//{attribute 'qualified_only'}
VAR_GLOBAL
	systemMethods : FB_System;
END_VAR

(* stored: Version 1.1.0.1, ProductVersion 3.1.4024.11
   GVL Misc: Id {b2366d92-2f76-473e-8c4c-cb3716fd6609} *)
